TYPE AxesMoveUnits :
(
	DEGREES := 0,
	RADIANS := 1,
	ARCSECONDS := 2
);
END_TYPE

(* stored: Version 1.1.0.1, ProductVersion 3.1.4019.2
   DUT AxesMoveUnits: Id {2f00a7ab-e827-4e96-834c-b7e8e3a259a2} *)
